TYPE NameHandle_t : Pointer to StrFileName_t; END_TYPE

(* stored: Version 1.1.0.1, ProductVersion 3.1.4024.12
   DUT NameHandle_t: Id {0248a818-a04e-4af0-b892-03fd9d1e4ccf} *)
